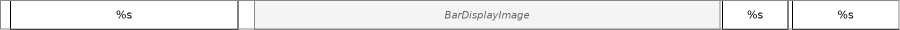
VISUALIZATION visuTaskData  // 900x30
VAR_IN_OUT
	d:typeIndividualTask; //data for faceplate
END_VAR
    Rectangle (10,0 228x30), "%s", text variable: d.singleTaskName, invisible if: NOT d.IsTaskEnabled
    BarDisplayImage (254,0 466x30), value: d.CycleTimeActual, invisible if: NOT d.IsTaskEnabled, style: BarDisplayImage-Gray, scale format: %.1f, scale 0..100
    Rectangle (792,0 107x30), "%s", invisible if: NOT d.IsTaskEnabled, text list: 'TaskText', text index: d.TaskStatus, colour variable: d.StateColour
    Rectangle (722,0 66x30), "%s", text variable: d.complexity, invisible if: NOT d.IsTaskEnabled, colour variable: d.StateColour
END_VISUALIZATION

(* stored: Version 1.1.0.1, ProductVersion 3.1.4024.12
   Visu visuTaskData: Id {80b0c714-4557-4275-98b6-85e01b2ad383} *)
